// SIMATIC S7-200 SMART project (STEP 7-Micro/WIN SMART), CPU SR30

SYMBOL_TABLE 风机和阀
温度量程下限           VD232
温度量程上限           VD228
模拟量最大值           VD216
模拟量最小值           VD208
压力量程下限           VD252
压力量程上限           VD268
风机停止             V2.0
风机启动             V2.1
风机远程             V2.2
风机故障             V2.3
风机输出             V2.4
风机               V2.5
风机运行反馈           V2.6
风机超时             V2.7
阀1停止             V3.0
阀1启动             V3.1
阀1远程             V3.2
阀1故障             V3.3
阀1输出             V3.4
阀1               V3.5
阀1运行反馈           V3.6
阀1超时             V3.7
阀2停止             V4.0
阀2启动             V4.1
阀2远程             V4.2
阀2故障             V4.3
阀2输出             V4.4
阀2               V4.5
阀2运行反馈           V4.6
阀2超时             V4.7
阀3停止             V5.0
阀3启动             V5.1
阀3远程             V5.2
阀3故障             V5.3
阀3输出             V5.4
阀3               V5.5
阀3运行反馈           V5.6
阀3超时             V5.7
阀4停止             V6.0
阀4启动             V6.1
阀4远程             V6.2
阀4故障             V6.3
阀4输出             V6.4
阀4               V6.5
阀4运行反馈           V6.6
阀4超时             V6.7
END_SYMBOL_TABLE

SYMBOL_TABLE 系统符号
Always_On        SM0.0    // 始终接通
END_SYMBOL_TABLE

SYMBOL_TABLE 点火烧嘴
点火命令1            V7.0
点火成功信号1          V7.1
故障复位1            V7.2
点火变压器1           V7.3
点火电磁阀1           V7.4
报警1              V7.5
空气压力1            V9.0
燃气压力1            V9.1
燃气泄漏             V9.2
允许点火1            V9.3
本地               V9.4
远程               V100.0
点火命令2            V7.6
点火成功信号2          V7.7
故障复位2            V8.0
点火变压器2           V8.1
点火电磁阀2           V8.2
报警2              V8.3
空气压力2            V9.6
燃气压力2            V9.7
允许点火2            V10.0
END_SYMBOL_TABLE

ORGANIZATION_BLOCK MAIN:OB1
TITLE=程序注释
BEGIN
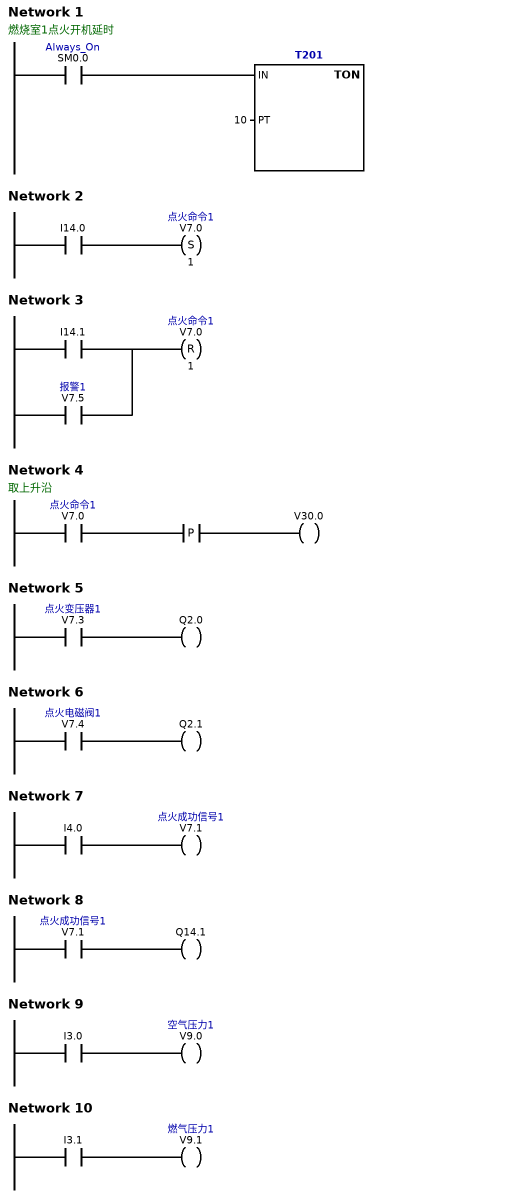
Network 1
// 燃烧室1点火开机延时
LD     Always_On:SM0.0
TON    T201, 10
Network 2
LD     I14.0
S      点火命令1:V7.0, 1
Network 3
LD     I14.1
O      报警1:V7.5
R      点火命令1:V7.0, 1
Network 4
// 取上升沿
LD     点火命令1:V7.0
EU
=      V30.0
Network 5
LD     点火变压器1:V7.3
=      Q2.0
Network 6
LD     点火电磁阀1:V7.4
=      Q2.1
Network 7
LD     I4.0
=      点火成功信号1:V7.1
Network 8
LD     点火成功信号1:V7.1
=      Q14.1
Network 9
LD     I3.0
=      空气压力1:V9.0
Network 10
LD     I3.1
=      燃气压力1:V9.1
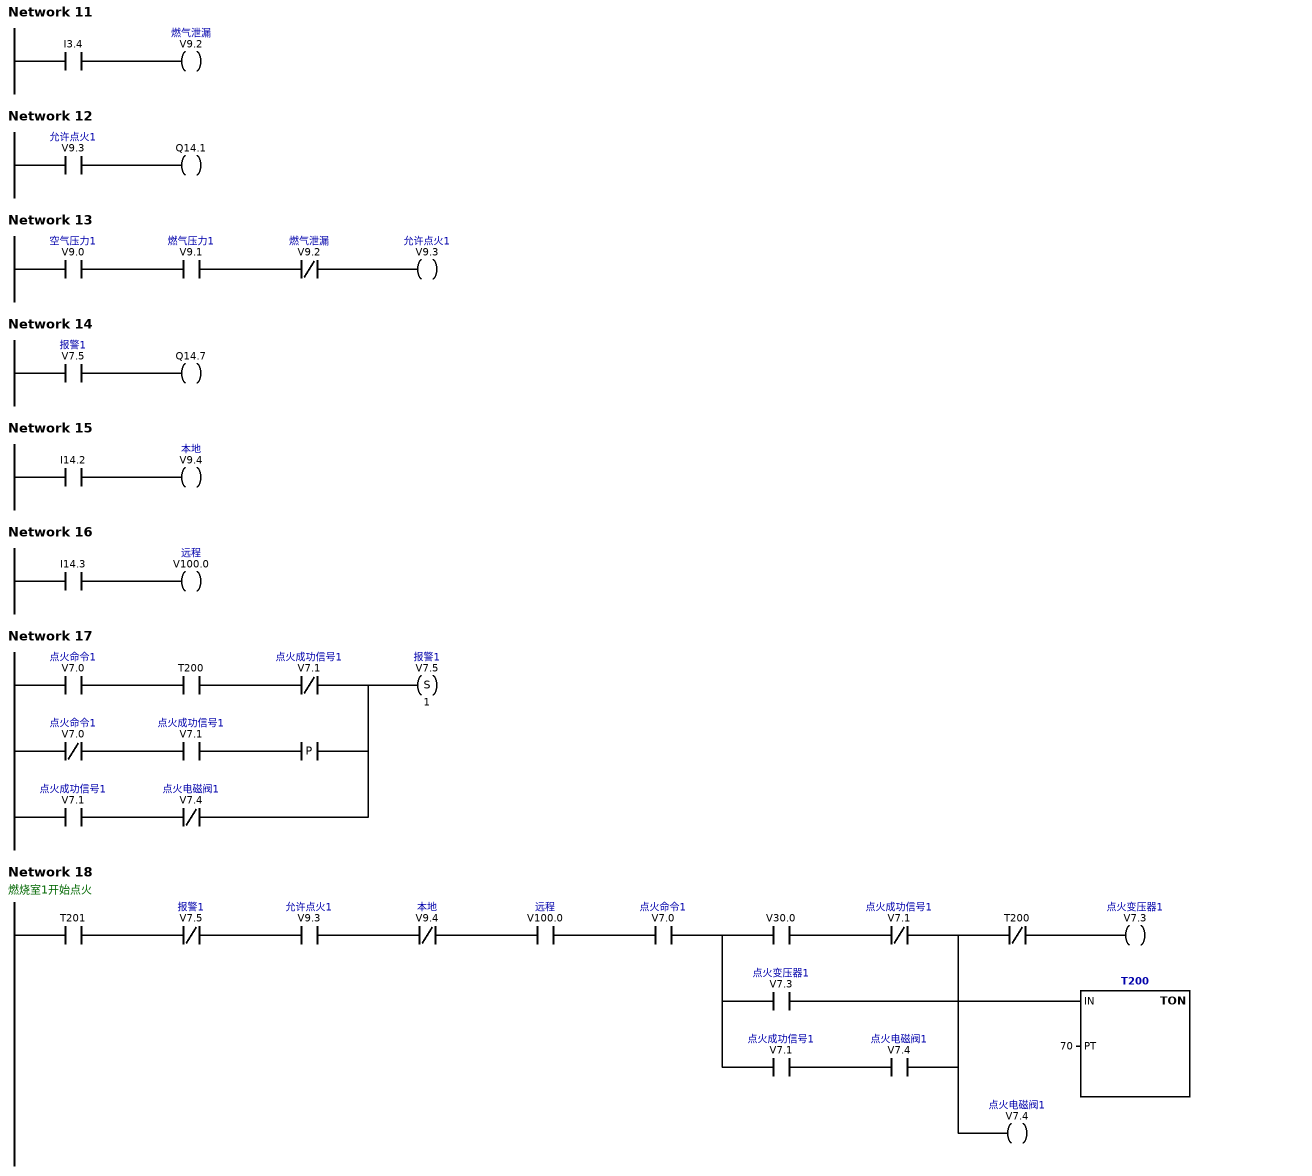
Network 11
LD     I3.4
=      燃气泄漏:V9.2
Network 12
LD     允许点火1:V9.3
=      Q14.1
Network 13
LD     空气压力1:V9.0
A      燃气压力1:V9.1
AN     燃气泄漏:V9.2
=      允许点火1:V9.3
Network 14
LD     报警1:V7.5
=      Q14.7
Network 15
// (network saved uncompiled; LAD cells follow)
// row 0: c0 -| |- I14.2  c1 -( ) 本地:V9.4
Network 16
// (network saved uncompiled; LAD cells follow)
// row 0: c0 -| |- I14.3  c1 -( ) 远程:V100.0
Network 17
LD     点火命令1:V7.0
A      T200
AN     点火成功信号1:V7.1
LDN    点火命令1:V7.0
A      点火成功信号1:V7.1
EU
OLD
LD     点火成功信号1:V7.1
AN     点火电磁阀1:V7.4
OLD
S      报警1:V7.5, 1
Network 18
// 燃烧室1开始点火
// (network saved uncompiled; LAD cells follow)
// row 0: c0 -| |- T201  c1 -|/|- 报警1:V7.5  c2 -| |- 允许点火1:V9.3  c3 -|/|- 本地:V9.4  c4 -| |- 远程:V100.0  c5 -| |- 点火命令1:V7.0 v  c6 -| |- V30.0  c7 -|/|- 点火成功信号1:V7.1 v  c8 -|/|- T200  c9 -( ) 点火变压器1:V7.3
// row 1: c5 ^v  c6 -| |- 点火变压器1:V7.3  c7 -- ^v  c8 --  c9 [TON T200 IN:=power@row1, PT:=70]
// row 2: c5 ^  c6 -| |- 点火成功信号1:V7.1  c7 -| |- 点火电磁阀1:V7.4 ^v  c9 [box]
// row 3: c7 ^  c8 -( ) 点火电磁阀1:V7.4
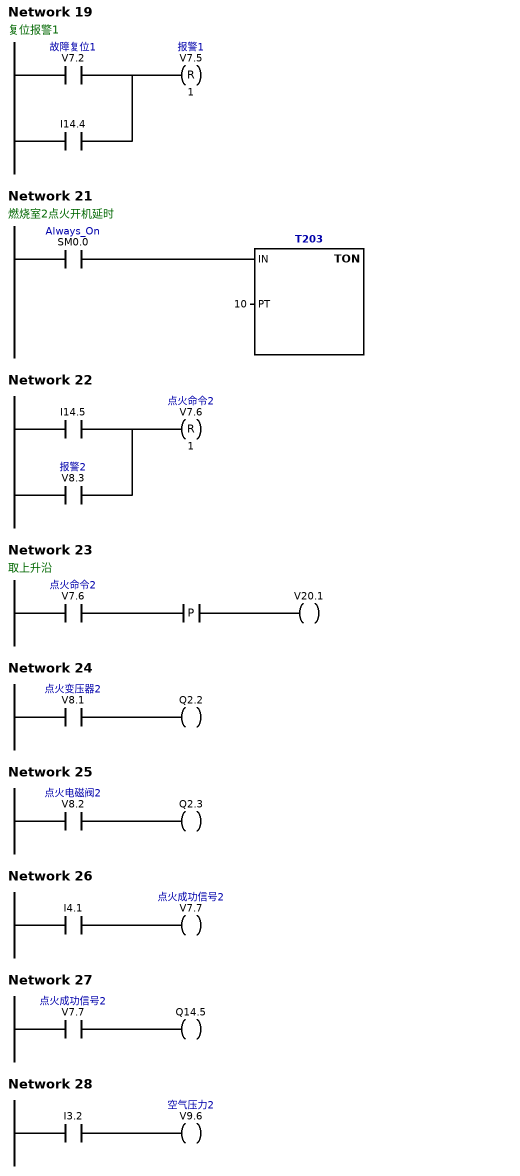
Network 19
// 复位报警1
LD     故障复位1:V7.2
O      I14.4
R      报警1:V7.5, 1
Network 21
// 燃烧室2点火开机延时
LD     Always_On:SM0.0
TON    T203, 10
Network 22
// (network saved uncompiled; LAD cells follow)
// row 0: c0 -| |- I14.5 v  c1 -(R) 点火命令2:V7.6, 1
// row 1: c0 -| |- 报警2:V8.3 ^
Network 23
// 取上升沿
LD     点火命令2:V7.6
EU
=      V20.1
Network 24
LD     点火变压器2:V8.1
=      Q2.2
Network 25
LD     点火电磁阀2:V8.2
=      Q2.3
Network 26
LD     I4.1
=      点火成功信号2:V7.7
Network 27
// (network saved uncompiled; LAD cells follow)
// row 0: c0 -| |- 点火成功信号2:V7.7  c1 -( ) Q14.5
Network 28
// (network saved uncompiled; LAD cells follow)
// row 0: c0 -| |- I3.2  c1 -( ) 空气压力2:V9.6
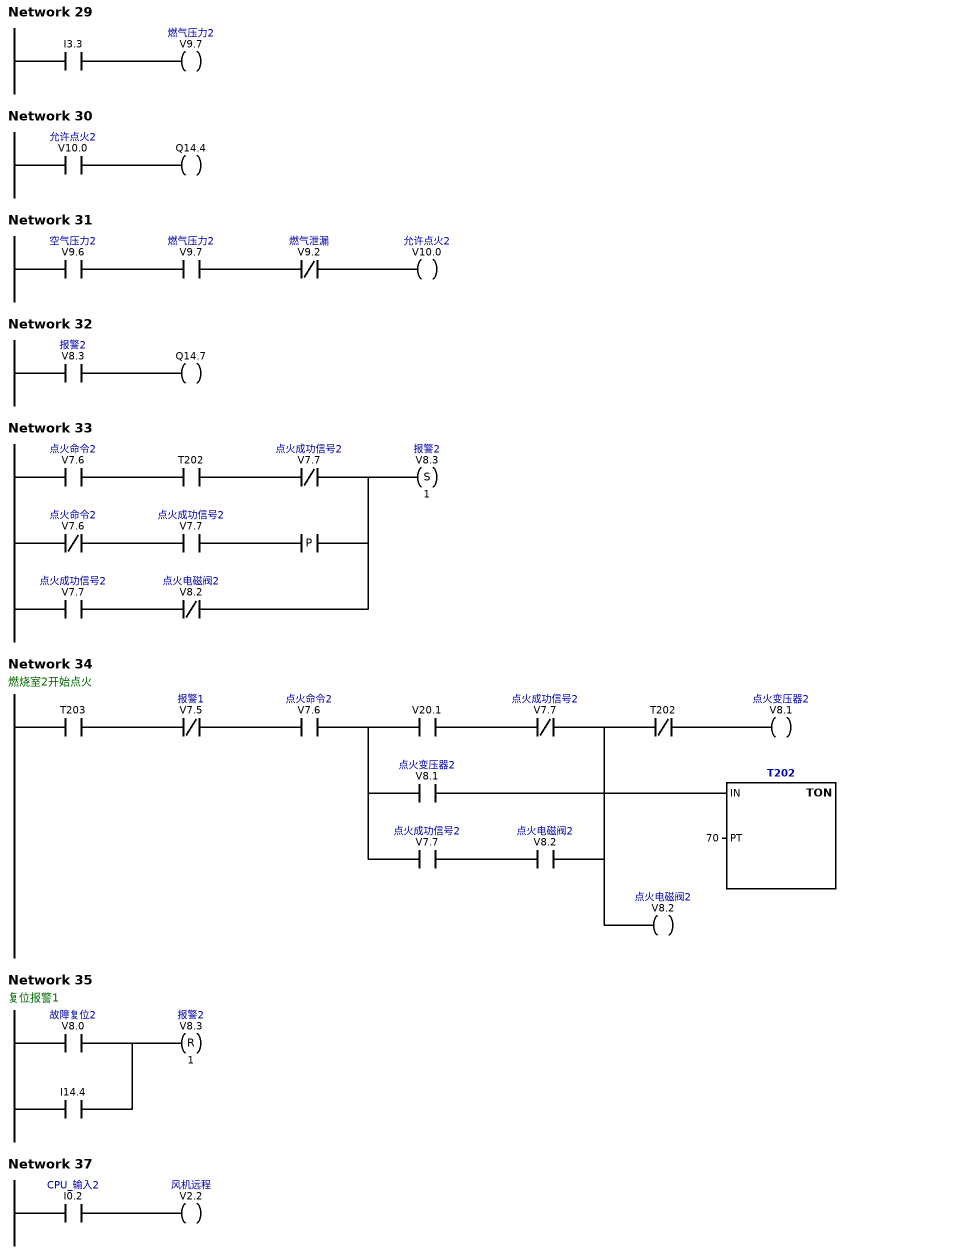
Network 29
// (network saved uncompiled; LAD cells follow)
// row 0: c0 -| |- I3.3  c1 -( ) 燃气压力2:V9.7
Network 30
// (network saved uncompiled; LAD cells follow)
// row 0: c0 -| |- 允许点火2:V10.0  c1 -( ) Q14.4
Network 31
// (network saved uncompiled; LAD cells follow)
// row 0: c0 -| |- 空气压力2:V9.6  c1 -| |- 燃气压力2:V9.7  c2 -|/|- 燃气泄漏:V9.2  c3 -( ) 允许点火2:V10.0
Network 32
// (network saved uncompiled; LAD cells follow)
// row 0: c0 -| |- 报警2:V8.3  c1 -( ) Q14.7
Network 33
// (network saved uncompiled; LAD cells follow)
// row 0: c0 -| |- 点火命令2:V7.6  c1 -| |- T202  c2 -|/|- 点火成功信号2:V7.7 v  c3 -(S) 报警2:V8.3, 1
// row 1: c0 -|/|- 点火命令2:V7.6  c1 -| |- 点火成功信号2:V7.7  c2 -|P|-  ^v
// row 2: c0 -| |- 点火成功信号2:V7.7  c1 -|/|- 点火电磁阀2:V8.2  c2 -- ^
Network 34
// 燃烧室2开始点火
LD     T203
AN     报警1:V7.5
A      点火命令2:V7.6
LD     V20.1
AN     点火成功信号2:V7.7
O      点火变压器2:V8.1
LD     点火成功信号2:V7.7
A      点火电磁阀2:V8.2
OLD
ALD
LPS
AN     T202
=      点火变压器2:V8.1
LRD
TON    T202, 70
LPP
=      点火电磁阀2:V8.2
Network 35
// 复位报警1
// (network saved uncompiled; LAD cells follow)
// row 0: c0 -| |- 故障复位2:V8.0 v  c1 -(R) 报警2:V8.3, 1
// row 1: c0 -| |- I14.4 ^
Network 37
LD     CPU_输入2:I0.2
=      风机远程:V2.2
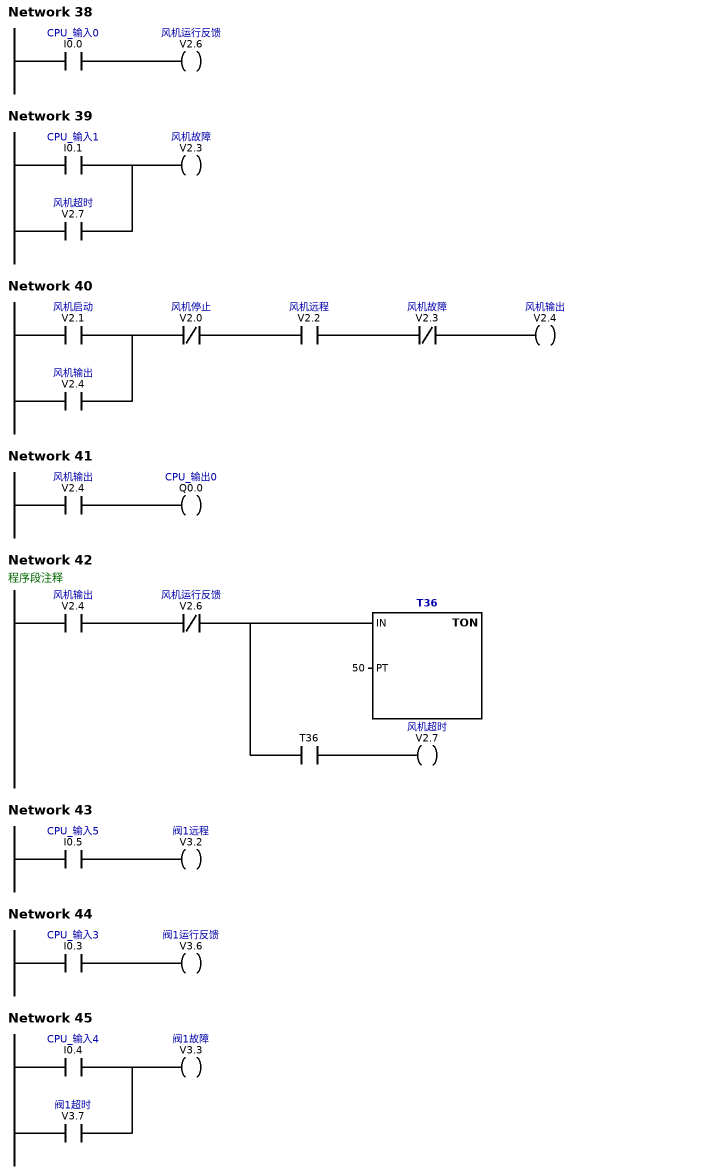
Network 38
LD     CPU_输入0:I0.0
=      风机运行反馈:V2.6
Network 39
LD     CPU_输入1:I0.1
O      风机超时:V2.7
=      风机故障:V2.3
Network 40
LD     风机启动:V2.1
O      风机输出:V2.4
AN     风机停止:V2.0
A      风机远程:V2.2
AN     风机故障:V2.3
=      风机输出:V2.4
Network 41
LD     风机输出:V2.4
=      CPU_输出0:Q0.0
Network 42
// 程序段注释
LD     风机输出:V2.4
AN     风机运行反馈:V2.6
TON    T36, 50
A      T36
=      风机超时:V2.7
Network 43
LD     CPU_输入5:I0.5
=      阀1远程:V3.2
Network 44
LD     CPU_输入3:I0.3
=      阀1运行反馈:V3.6
Network 45
LD     CPU_输入4:I0.4
O      阀1超时:V3.7
=      阀1故障:V3.3
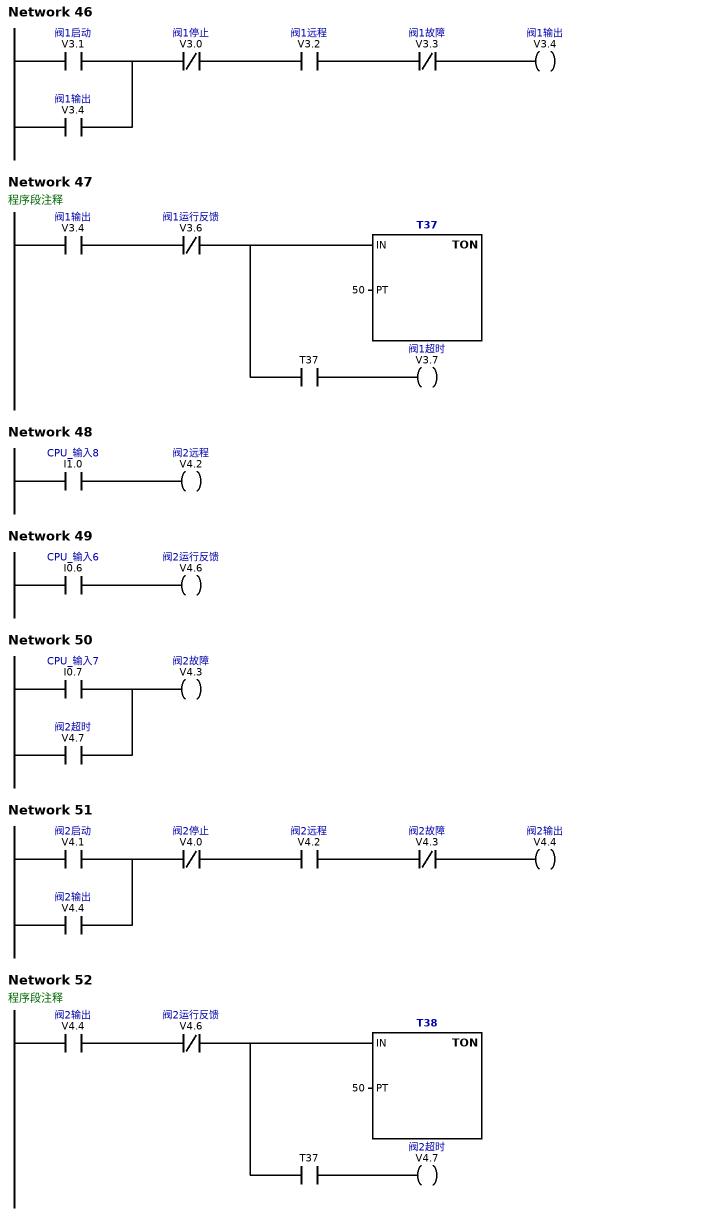
Network 46
LD     阀1启动:V3.1
O      阀1输出:V3.4
AN     阀1停止:V3.0
A      阀1远程:V3.2
AN     阀1故障:V3.3
=      阀1输出:V3.4
Network 47
// 程序段注释
LD     阀1输出:V3.4
AN     阀1运行反馈:V3.6
TON    T37, 50
A      T37
=      阀1超时:V3.7
Network 48
LD     CPU_输入8:I1.0
=      阀2远程:V4.2
Network 49
LD     CPU_输入6:I0.6
=      阀2运行反馈:V4.6
Network 50
LD     CPU_输入7:I0.7
O      阀2超时:V4.7
=      阀2故障:V4.3
Network 51
LD     阀2启动:V4.1
O      阀2输出:V4.4
AN     阀2停止:V4.0
A      阀2远程:V4.2
AN     阀2故障:V4.3
=      阀2输出:V4.4
Network 52
// 程序段注释
LD     阀2输出:V4.4
AN     阀2运行反馈:V4.6
TON    T38, 50
A      T37
=      阀2超时:V4.7
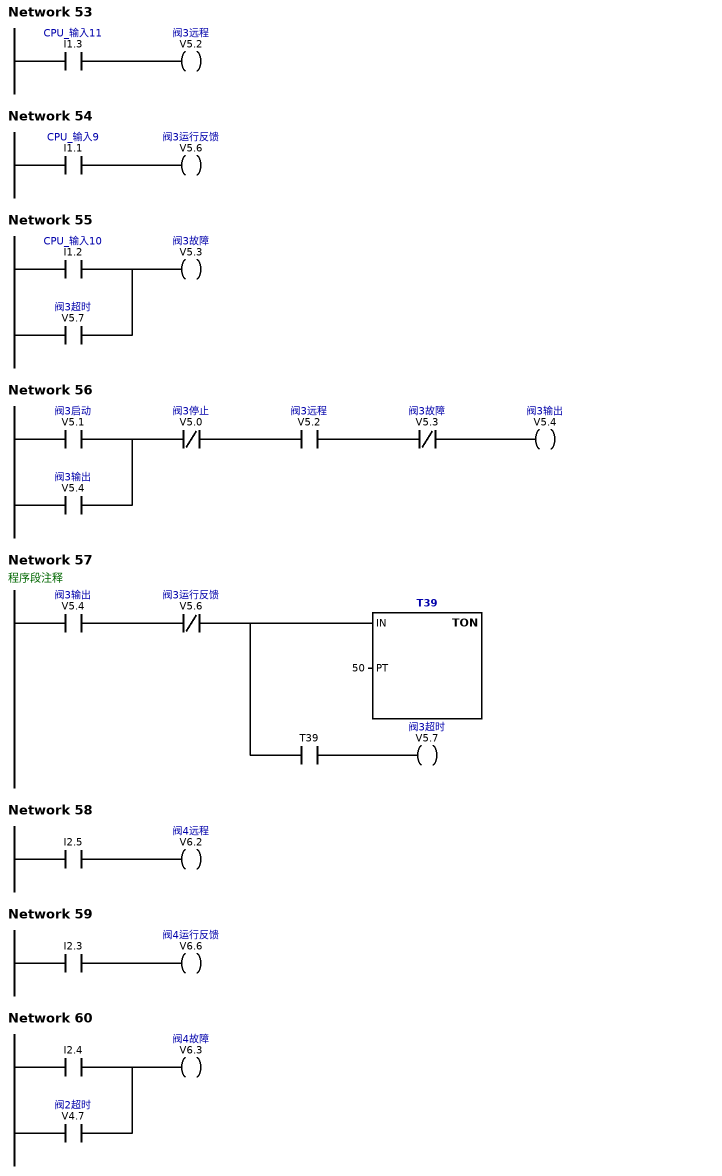
Network 53
LD     CPU_输入11:I1.3
=      阀3远程:V5.2
Network 54
LD     CPU_输入9:I1.1
=      阀3运行反馈:V5.6
Network 55
LD     CPU_输入10:I1.2
O      阀3超时:V5.7
=      阀3故障:V5.3
Network 56
LD     阀3启动:V5.1
O      阀3输出:V5.4
AN     阀3停止:V5.0
A      阀3远程:V5.2
AN     阀3故障:V5.3
=      阀3输出:V5.4
Network 57
// 程序段注释
LD     阀3输出:V5.4
AN     阀3运行反馈:V5.6
TON    T39, 50
A      T39
=      阀3超时:V5.7
Network 58
LD     I2.5
=      阀4远程:V6.2
Network 59
LD     I2.3
=      阀4运行反馈:V6.6
Network 60
LD     I2.4
O      阀2超时:V4.7
=      阀4故障:V6.3
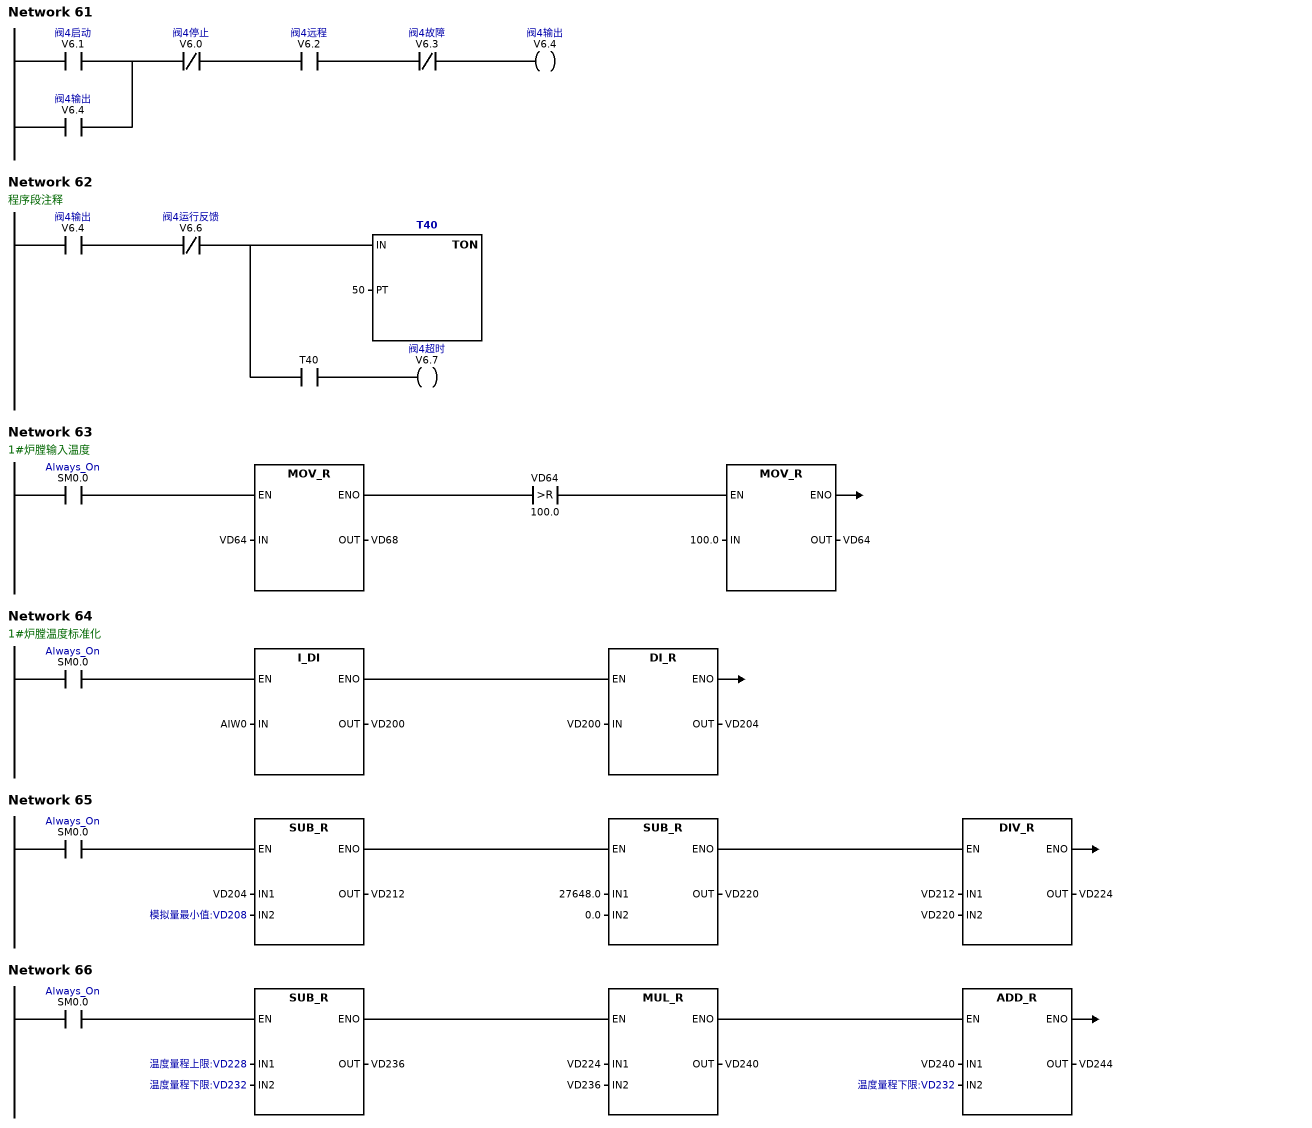
Network 61
LD     阀4启动:V6.1
O      阀4输出:V6.4
AN     阀4停止:V6.0
A      阀4远程:V6.2
AN     阀4故障:V6.3
=      阀4输出:V6.4
Network 62
// 程序段注释
LD     阀4输出:V6.4
AN     阀4运行反馈:V6.6
TON    T40, 50
A      T40
=      阀4超时:V6.7
Network 63
// 1#炉膛输入温度
LD     Always_On:SM0.0
MOVR   VD64, VD68
AENO
AR>    VD64, 100.0
MOVR   100.0, VD64
Network 64
// 1#炉膛温度标准化
LD     Always_On:SM0.0
ITD    AIW0, VD200
AENO
DTR    VD200, VD204
Network 65
LD     Always_On:SM0.0
MOVR   VD204, VD212
AENO
-R     模拟量最小值:VD208, VD212
AENO
MOVR   27648.0, VD220
AENO
-R     0.0, VD220
AENO
MOVR   VD212, VD224
/R     VD220, VD224
Network 66
LD     Always_On:SM0.0
MOVR   温度量程上限:VD228, VD236
AENO
-R     温度量程下限:VD232, VD236
AENO
MOVR   VD224, VD240
AENO
*R     VD236, VD240
AENO
MOVR   VD240, VD244
+R     温度量程下限:VD232, VD244
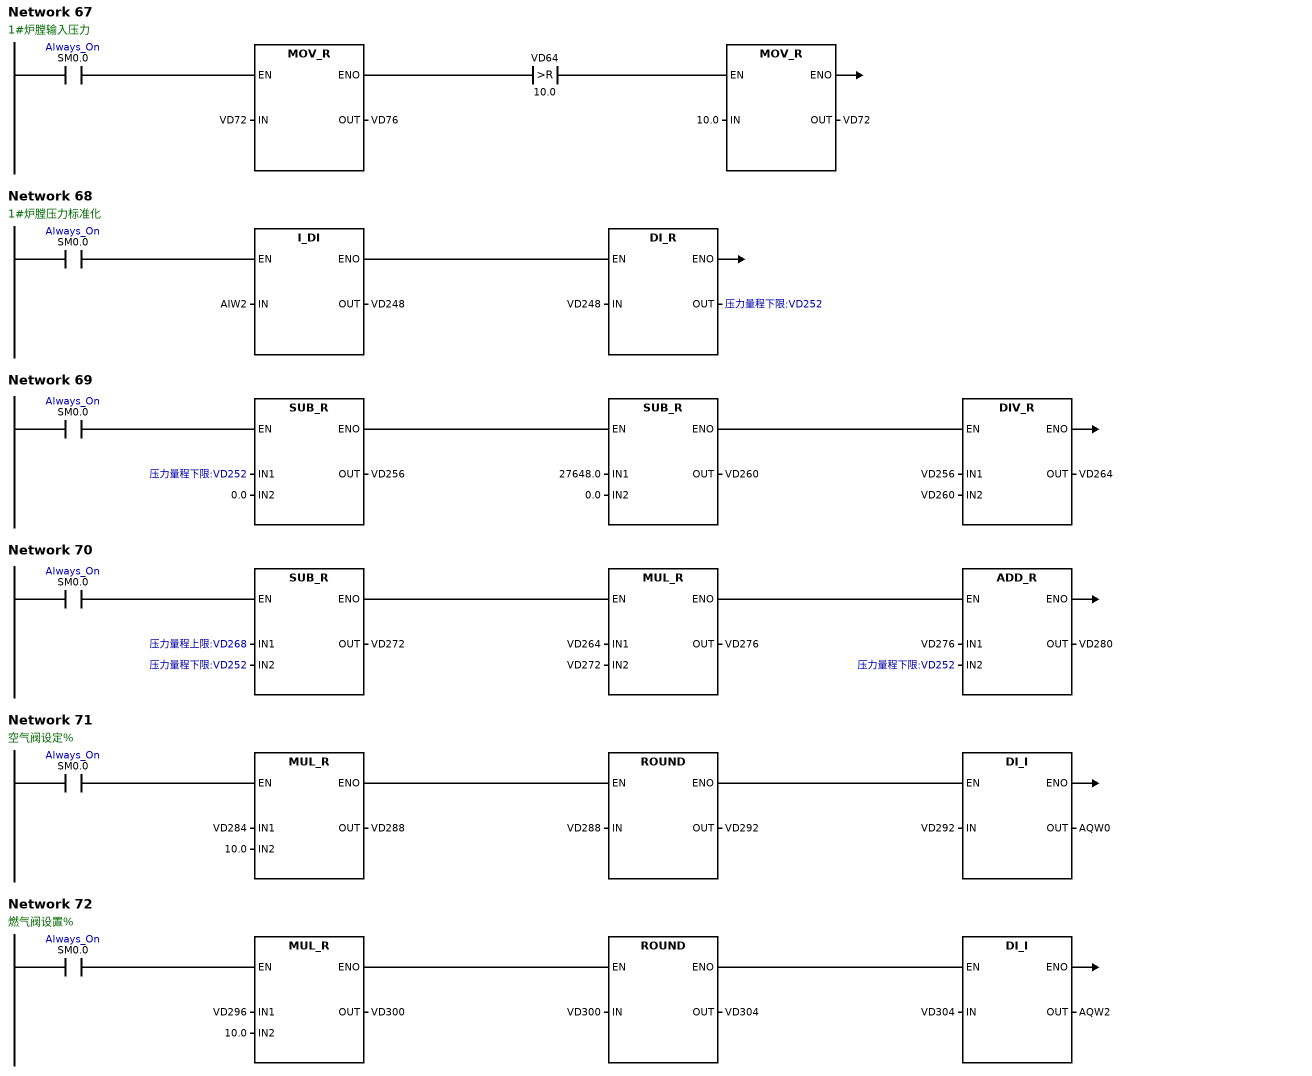
Network 67
// 1#炉膛输入压力
LD     Always_On:SM0.0
MOVR   VD72, VD76
AENO
AR>    VD64, 10.0
MOVR   10.0, VD72
Network 68
// 1#炉膛压力标准化
LD     Always_On:SM0.0
ITD    AIW2, VD248
AENO
DTR    VD248, 压力量程下限:VD252
Network 69
LD     Always_On:SM0.0
MOVR   压力量程下限:VD252, VD256
AENO
-R     0.0, VD256
AENO
MOVR   27648.0, VD260
AENO
-R     0.0, VD260
AENO
MOVR   VD256, VD264
/R     VD260, VD264
Network 70
LD     Always_On:SM0.0
MOVR   压力量程上限:VD268, VD272
AENO
-R     压力量程下限:VD252, VD272
AENO
MOVR   VD264, VD276
AENO
*R     VD272, VD276
AENO
MOVR   VD276, VD280
+R     压力量程下限:VD252, VD280
Network 71
// 空气阀设定%
LD     Always_On:SM0.0
MOVR   VD284, VD288
AENO
*R     10.0, VD288
AENO
ROUND  VD288, VD292
AENO
DTI    VD292, AQW0
Network 72
// 燃气阀设置%
LD     Always_On:SM0.0
MOVR   VD296, VD300
AENO
*R     10.0, VD300
AENO
ROUND  VD300, VD304
AENO
DTI    VD304, AQW2
END_ORGANIZATION_BLOCK

// SBR1: protected block, not included

// SBR2: protected block, not included

// SBR3: protected block, not included

// SBR4: protected block, not included

// SBR5: protected block, not included

// SBR6: protected block, not included

// SBR7: protected block, not included
